FUNCTION_BLOCK FB_OneShotExample
VAR
	execute : BOOL;
END_VAR

M_OneShot(execute);

METHOD M_OneShot

VAR_INPUT
	_execute : BOOL;
END_VAR

VAR_INST
	execTrig : R_Trig;
END_VAR
execTrig(CLK := _execute);
RETURN (NOT execTrig.Q);

// Do code here, will only be called for each time _execute does from low to high
END_METHOD

END_FUNCTION_BLOCK

(* stored: Version 1.1.0.1
   POU FB_OneShotExample: Id {ecd4cb75-baed-475e-950b-0e9effe618c7}, SpecialFunc None
   Method M_OneShot: Id {754dceb4-eb65-49ed-95da-4c10edb29040} *)
